PROGRAM Rotina020
VAR
	status: INT;
	
	posicaoAtual: STRING;
	envialog: STRING;
	
	fbTimeVentila: ton;
	fbTimeAqueci: ton;
	
	a: INT;
END_VAR

fbTimeVentila();
fbTimeAqueci();
a:=1;

CASE status OF

0:
IF gvl_p.arrStatusEstufas[a].start AND STRING_TO_DT(gvl.progInicio[a]) <= systemtime_to_dt(gvl.fbGetLocalSystemTime.systemTime)  THEN
	status:= 5;
	
	gvl.bstartchart020:= TRUE;
	gvl_p.zona1setpt_020:= gvl_p.arrStatusEstufas[a].tempSeca;
	gvl_p.zona2setpt_020:= gvl_p.arrStatusEstufas[a].tempSeca;
	gvl.liga_ventilacao_020:= TRUE;
	fbTimeVentila(in:= TRUE, pt:=T#1S);
	
	gvl_p.etapa_process[a] := 'Inicializando';
	
ELSE
	status:= 0;
	IF gvl_p.arrStatusEstufas[a].start THEN
		gvl_p.etapa_process[a] := gvl.progInicio[a];
	END_IF
END_IF
5:
IF fbTimeVentila.Q THEN
	status:= 10;
	gvl.liga_ventilacao_020:=FALSE;
	fbTimeVentila(in:= FALSE);
ELSE
	status:= 5;
END_IF

10:
IF gvl.ventilacao_Ligada_020 THEN
	status:= 15;
	
	gvl.liga_aquecimento_020:= TRUE;
	fbTimeAqueci(in:= TRUE, pt:= T#1S);
	
	gvl_p.etapa_process[a] := 'Aquecendo';
	
ELSE
	status:= 10;
END_IF

15:
IF fbTimeAqueci.Q THEN
	status:= 20;
	
	gvl.liga_aquecimento_020:= FALSE;
	fbTimeAqueci(in:=false);
ELSE
	status:= 15;
END_IF

20:
IF gvl.zona1atual_020 >= gvl_p.zona1setpt_020 THEN
	status:= 30;

gvl.progInicio[a]:= DT_TO_STRING(gvl.somaTempo);
	
///// CALCULAR FIM DA SECAGEM E DA ARMAZENAGEM --------------------------------------------------------------------------------
gvl_p.arrStatusEstufas[a].inicioSecagem := STRING_TO_DT(gvl.progInicio[a]);
gvl_p.arrStatusEstufas[a].fimSecagem := STRING_TO_DT(gvl.progInicio[a]) + gvl_p.arrStatusEstufas[a].tempoSecagem;
gvl_P.arrStatusEstufas[a].prevFimSeca := gvl_p.arrStatusEstufas[a].fimSecagem;
gvl_p.arrStatusEstufas[a].fimArmazenagem := gvl_p.arrStatusEstufas[a].fimSecagem + gvl_p.arrStatusEstufas[a].tempoArmazenagem ;

///// IMPRIMIR A HORA E A DATA DO INICIO DA SECAGEM ---------------------------------------------------------------------------
gvl_p.arrStatusEstufas[a].statusInicioSecagem := '';
gvl_p.arrStatusEstufas[a].statusInicioSecagem := concat(gvl_p.arrStatusEstufas[a].statusInicioSecagem,gvl.hora);
gvl_p.arrStatusEstufas[a].statusInicioSecagem := concat(gvl_p.arrStatusEstufas[a].statusInicioSecagem,':');
gvl_p.arrStatusEstufas[a].statusInicioSecagem := concat(gvl_p.arrStatusEstufas[a].statusInicioSecagem,gvl.minuto);
gvl_p.arrStatusEstufas[a].statusInicioSecagem := concat(gvl_p.arrStatusEstufas[a].statusInicioSecagem,' ');
gvl_p.arrStatusEstufas[a].statusInicioSecagem := concat(gvl_p.arrStatusEstufas[a].statusInicioSecagem,gvl.dia);
gvl_p.arrStatusEstufas[a].statusInicioSecagem := concat(gvl_p.arrStatusEstufas[a].statusInicioSecagem,'/');
gvl_p.arrStatusEstufas[a].statusInicioSecagem := concat(gvl_p.arrStatusEstufas[a].statusInicioSecagem,gvl.mes);
gvl_p.arrStatusEstufas[a].statusInicioSecagem := concat(gvl_p.arrStatusEstufas[a].statusInicioSecagem,'/');
gvl_p.arrStatusEstufas[a].statusInicioSecagem := concat(gvl_p.arrStatusEstufas[a].statusInicioSecagem,gvl.ano);

//--------------------REATOR------------------------------------

IF gravarConfigPosicao_Reator.bGravarConfigPosicao_Reator THEN
	gvl_p.arrStatusEstufas[a].inicioReator := '';
	gvl_p.arrStatusEstufas[a].inicioReator := concat(gvl_p.arrStatusEstufas[a].inicioReator,gvl.hora);
	gvl_p.arrStatusEstufas[a].inicioReator := concat(gvl_p.arrStatusEstufas[a].inicioReator,':');
	gvl_p.arrStatusEstufas[a].inicioReator := concat(gvl_p.arrStatusEstufas[a].inicioReator,gvl.minuto);
	gvl_p.arrStatusEstufas[a].inicioReator := concat(gvl_p.arrStatusEstufas[a].inicioReator,' ');
	gvl_p.arrStatusEstufas[a].inicioReator := concat(gvl_p.arrStatusEstufas[a].inicioReator,gvl.dia);
	gvl_p.arrStatusEstufas[a].inicioReator := concat(gvl_p.arrStatusEstufas[a].inicioReator,'/');
	gvl_p.arrStatusEstufas[a].inicioReator := concat(gvl_p.arrStatusEstufas[a].inicioReator,gvl.mes);
	gvl_p.arrStatusEstufas[a].inicioReator := concat(gvl_p.arrStatusEstufas[a].inicioReator,'/');
	gvl_P.arrStatusEstufas[a].inicioReator := concat(gvl_p.arrStatusEstufas[a].inicioReator,gvl.ano);
END_IF

///// DECOMPOR A VARIAVEL FIM DA SECAGEM -----------------------------------------------------------------------------------------------
gvl_p.arrStatusEstufas[a].diaSec := MID(STR:= DT_TO_STRING(gvl_p.arrStatusEstufas[a].fimSecagem) , LEN:= 2, POS:=12);
gvl_p.arrStatusEstufas[a].mesSec := MID(STR:= DT_TO_STRING(gvl_p.arrStatusEstufas[a].fimSecagem), LEN:= 2, POS:=9);
gvl_p.arrStatusEstufas[a].anoSec := MID(STR:= DT_TO_STRING(gvl_p.arrStatusEstufas[a].fimSecagem), LEN:= 2, POS:=6);
gvl_p.arrStatusEstufas[a].horaSec := MID(STR:= DT_TO_STRING(gvl_p.arrStatusEstufas[a].fimSecagem), LEN:= 2, POS:=15);
gvl_p.arrStatusEstufas[a].minutoSec := MID(STR:= DT_TO_STRING(gvl_p.arrStatusEstufas[a].fimSecagem), LEN:= 2, POS:=18);

///// IMPRIMIR A HORA E A DATA DO FIM DA SECAGEM --------------------------------------------------------------------------------------------------------
gvl_p.arrStatusEstufas[a].statusFimSecagem := '';
gvl_p.arrStatusEstufas[a].statusFimSecagem := concat(gvl_p.arrStatusEstufas[a].statusFimSecagem,gvl_p.arrStatusEstufas[a].horaSec);
gvl_p.arrStatusEstufas[a].statusFimSecagem := concat(gvl_p.arrStatusEstufas[a].statusFimSecagem,':');
gvl_p.arrStatusEstufas[a].statusFimSecagem := concat(gvl_p.arrStatusEstufas[a].statusFimSecagem,gvl_p.arrStatusEstufas[a].minutoSec);
gvl_p.arrStatusEstufas[a].statusFimSecagem := concat(gvl_p.arrStatusEstufas[a].statusFimSecagem,' ');
gvl_p.arrStatusEstufas[a].statusFimSecagem := concat(gvl_p.arrStatusEstufas[a].statusFimSecagem,gvl_p.arrStatusEstufas[a].diaSec);
gvl_p.arrStatusEstufas[a].statusFimSecagem := concat(gvl_p.arrStatusEstufas[a].statusFimSecagem,'/');
gvl_p.arrStatusEstufas[a].statusFimSecagem := concat(gvl_p.arrStatusEstufas[a].statusFimSecagem,gvl_p.arrStatusEstufas[a].mesSec);
gvl_p.arrStatusEstufas[a].statusFimSecagem := concat(gvl_p.arrStatusEstufas[a].statusFimSecagem,'/');
gvl_p.arrStatusEstufas[a].statusFimSecagem := concat(gvl_p.arrStatusEstufas[a].statusFimSecagem,gvl_p.arrStatusEstufas[a].anoSec);

///// DECOMPOR A VARIAVEL FIM DA ARMAZENAGEM -------------------------------------------------------------------------------------------
gvl_p.arrStatusEstufas[a].diaArm := MID(STR:= DT_TO_STRING(gvl_p.arrStatusEstufas[a].fimArmazenagem) , LEN:= 2, POS:=12);
gvl_p.arrStatusEstufas[a].mesArm := MID(STR:= DT_TO_STRING(gvl_p.arrStatusEstufas[a].fimArmazenagem), LEN:= 2, POS:=9);
gvl_p.arrStatusEstufas[a].anoArm := MID(STR:= DT_TO_STRING(gvl_P.arrStatusEstufas[a].fimArmazenagem), LEN:= 2, POS:=6);
gvl_p.arrStatusEstufas[a].horaArm := MID(STR:= DT_TO_STRING(gvl_P.arrStatusEstufas[a].fimArmazenagem), LEN:= 2, POS:=15);
gvl_p.arrStatusEstufas[a].minutoArm := MID(STR:= DT_TO_STRING(gvl_p.arrStatusEstufas[a].fimArmazenagem), LEN:= 2, POS:=18);

///// IMPRIMIR A HORA E A DATA DO FIM DA ARMAZENAGEM -----------------------------------------------------------------------------------------------------------
gvl_p.arrStatusEstufas[a].statusFimArmazenagem := '';
gvl_p.arrStatusEstufas[a].statusFimArmazenagem := concat(gvl_p.arrStatusEstufas[a].statusFimArmazenagem,gvl_p.arrStatusEstufas[a].horaArm);
gvl_p.arrStatusEstufas[a].statusFimArmazenagem := concat(gvl_p.arrStatusEstufas[a].statusFimArmazenagem,':');
gvl_p.arrStatusEstufas[a].statusFimArmazenagem := concat(gvl_p.arrStatusEstufas[a].statusFimArmazenagem,gvl_p.arrStatusEstufas[a].minutoArm);
gvl_p.arrStatusEstufas[a].statusFimArmazenagem := concat(gvl_p.arrStatusEstufas[a].statusFimArmazenagem,' ');
gvl_p.arrStatusEstufas[a].statusFimArmazenagem := concat(gvl_p.arrStatusEstufas[a].statusFimArmazenagem,gvl_p.arrStatusEstufas[a].diaArm);
gvl_p.arrStatusEstufas[a].statusFimArmazenagem := concat(gvl_p.arrStatusEstufas[a].statusFimArmazenagem,'/');
gvl_p.arrStatusEstufas[a].statusFimArmazenagem := concat(gvl_p.arrStatusEstufas[a].statusFimArmazenagem,gvl_p.arrStatusEstufas[a].mesArm);
gvl_p.arrStatusEstufas[a].statusFimArmazenagem := concat(gvl_p.arrStatusEstufas[a].statusFimArmazenagem,'/');
gvl_p.arrStatusEstufas[a].statusFimArmazenagem := concat(gvl_p.arrStatusEstufas[a].statusFimArmazenagem,gvl_p.arrStatusEstufas[a].anoArm);

///// GERADOR DE LOG -------------------------------------------------------------
envialog:= 'Programação Iniciada ESTUFA 1';
gvl.logRegister20:= envialog;

gvl_p.etapa_process[a] := 'Secagem';

ELSE
	status:= 20;
END_IF

30:
IF gvl_p.arrStatusEstufas[a].prevFimSeca = systemtime_to_dt(gvl.fbGetLocalSystemTime.systemTime) THEN
	status:= 40;
	
	gvl.zona1atual_020:= gvl_p.arrStatusEstufas[a].tempArm;
	gvl.zona2atual_020:= gvl_p.arrStatusEstufas[a].tempArm;
	
///// GERADOR DE LOG -------------------------------------------------------------
envialog:= 'Armazenagem Iniciada ESTUFA 1';
gvl.logRegister20:= envialog;
	
gvl_p.etapa_process[a] := 'Armazenagem';

ELSE
	status:= 30;
END_IF

40:
IF gvl_p.arrStatusEstufas[a].fimArmazenagem = systemtime_to_dt(gvl.fbGetLocalSystemTime.systemTime) THEN
	status:= 50;
	
	gvl_p.arrStatusEstufas[a].start:= FALSE;
	gvl.bstartchart020:= FALSE;
	gvl.desl_aquecimento_020:= TRUE;
	fbTimeAqueci(in:=TRUE, pt:=T#1S);
	
	gvl_p.etapa_process[a] := '';
	
	gvl_p.arrStatusEstufas[a].statusInicioSecagem := '';
	gvl_p.arrStatusEstufas[a].inicioReator := '';
	gvl_p.arrStatusEstufas[a].statusFimSecagem := '';
	gvl_p.arrStatusEstufas[a].statusFimArmazenagem := '';
	gvl_p.arrStatusEstufas[a].fimSecagem:= DT#1970-1-1-0:0:0;
	
	
///// GERADOR DE LOG -------------------------------------------------------------
envialog:= 'Programação Finalizada ESTUFA 1';
gvl.logRegister20:= envialog;

ELSE
	status:= 40;
END_IF

45:
IF gvl_p.arrStatusEstufas[a].start THEN
status:= 50;
	
	gvl_p.arrStatusEstufas[a].start:= FALSE;
	gvl.bstartchart020:= FALSE;
	gvl.desl_aquecimento_020:= TRUE;
	fbTimeAqueci(in:=TRUE, pt:=T#1S);
	
	gvl_p.etapa_process[a] := '';
	
	gvl_p.arrStatusEstufas[a].statusInicioSecagem := '';
	gvl_p.arrStatusEstufas[a].inicioReator := '';
	gvl_p.arrStatusEstufas[a].statusFimSecagem := '';
	gvl_p.arrStatusEstufas[a].statusFimArmazenagem := '';
	gvl_p.arrStatusEstufas[a].fimSecagem:= DT#1970-1-1-0:0:0;
	
	
///// GERADOR DE LOG -------------------------------------------------------------
envialog:= 'Programação Finalizada ESTUFA 1';
gvl.logRegister20:= envialog;
ELSE
	status:= 45;
END_IF

50:
IF fbTimeAqueci.Q THEN
	status:= 0;
	
	gvl.desl_aquecimento_020:= FALSE;
	fbTimeAqueci(in:= FALSE);
	
ELSE
	status:= 50;
END_IF
END_CASE

END_PROGRAM

(* stored: Version 1.1.0.1, ProductVersion 3.1.4024.12
   POU Rotina020: Id {c4be85a0-018a-4a19-a152-e8cf438ae634}, SpecialFunc None *)
